Yaskawa INFORM job: R1_72,2(0,0)KM-OK.JBI

/JOB
//NAME R1_72,2(0,0)KM-OK
///FOLDERNAME KRIS-SCIANA
//POS
///NPOS 76,76,0,3,0,0
///TOOL 0
///POSTYPE PULSE
///PULSE
C00000=-88252,73272,-8021,3471,94135,-39741
C00001=-196921,-21278,-79002,-15523,92407,23647
C00002=-191529,-10180,-72050,-27767,99083,38733
C00003=-191529,-10180,-72050,-27767,99083,38733
C00004=-206105,-1744,-8023,-24853,79126,31669
C00005=-210790,-9435,-14216,-24034,77614,30226
C00006=-211112,-7151,-9678,-24113,76035,30431
C00007=-211112,-6884,-8412,-24172,75449,30554
C00008=-211112,-7143,-9634,-24115,76015,30436
C00009=-211447,-5344,-8192,-24050,75949,30323
C00010=-211112,-7143,-9634,-24115,76015,30436
C00011=-203899,-948,-19131,-24926,86387,30960
C00012=-203899,16721,-46212,-27001,109725,25798
C00013=-213997,-36135,-90156,-18508,92135,33607
C00014=-215703,-40125,-89891,-17749,89721,33477
C00015=-216394,-41642,-89732,-17450,88761,33414
C00016=-216190,-46458,-89537,-17546,86322,33825
C00017=-216581,-43974,-88082,-17376,86615,33666
C00018=-216757,-44589,-88447,-17302,86492,33627
C00019=-216394,-41642,-89732,-17450,88761,33414
C00020=-215410,-41044,-89232,-17867,88937,33676
C00021=-215562,-42319,-88713,-17803,87979,33772
C00022=-215410,-41044,-89232,-17867,88937,33676
C00023=-216394,-41642,-89732,-17450,88761,33414
C00024=-200348,-21688,-81312,-31633,113980,39480
C00025=-200646,-25016,-80489,-31008,111986,39985
C00026=-201612,-26033,-81353,-30788,111712,39736
C00027=-200646,-25016,-80489,-31008,111986,39985
C00028=-200348,-21688,-81312,-31633,113980,39480
C00029=-204378,-25649,-84759,-30672,112905,38454
C00030=-203466,-23371,-84449,-31149,114010,38425
C00031=-201237,-17494,-83481,-32404,116710,38313
C00032=-183775,-3850,-69382,-22164,99452,52082
C00033=-187139,105474,25900,5524,97478,-74523
C00034=-183987,78008,14988,-30780,97915,-53143
C00035=-185860,79679,21494,-38294,98804,-45722
C00036=-187540,86449,24962,5600,88344,-75041
C00037=-187072,89119,27221,5424,88298,-74904
C00038=-185446,79208,21072,-38405,98978,-45626
C00039=-185286,79610,21498,-38440,98994,-45572
C00040=-184095,83249,26388,-38603,98564,-44953
C00041=-184985,79410,21976,-38469,98802,-45386
C00042=-185085,78027,18507,-38623,99890,-45822
C00043=-184563,78672,15161,-39118,101977,-46400
C00044=-123480,133166,88670,-6552,116959,-64608
C00045=-123480,133166,88670,-6552,116959,-64608
C00046=-92269,117134,36709,3424,120351,-70294
C00047=-88374,116940,55217,-2527,120928,-72150
C00048=-88375,114548,55776,-2482,119356,-72114
C00049=-88651,123794,71043,-488,118252,-71721
C00050=-88408,114754,56297,-2480,119142,-72120
C00051=-88628,116331,59860,-2466,117754,-72169
C00052=-88954,122720,69576,-537,118600,-71834
C00053=-90233,119037,64628,-750,119747,-72317
C00054=-98563,95834,34419,17716,116287,-71642
C00055=-98641,94945,33315,17755,116515,-71636
C00056=-98178,89163,25359,18092,118260,-71172
C00057=-93588,99005,30718,8872,122903,-71358
C00058=-94574,131390,74567,2575,121590,-32143
C00059=-94435,131728,75046,2064,81257,-32153
C00060=-94150,154511,102675,2539,39785,-31487
C00061=-125444,148323,76798,-7366,54308,24231
C00062=-94150,154507,102675,2551,39784,-31488
C00063=-139725,-91160,-117526,-40600,105870,54843
C00064=-191529,-10180,-72050,-27767,99083,38733
C00065=-206105,-1744,-8023,-24853,79126,31669
C00066=-208371,-7084,-12355,-24468,78381,30975
C00067=-208875,-4028,-7246,-24508,76793,31119
C00068=-211010,-1092,-5442,-21718,78200,30111
C00069=-214621,-3970,-7511,-21112,77073,28985
C00070=-213962,-6039,-9919,-21200,77633,29128
C00071=-208371,-7084,-12355,-24468,78381,30975
C00072=-191529,-10180,-72050,-27767,99083,38733
C00073=-132846,-97761,-120048,-41164,107386,57132
C00074=-122033,25891,-66087,-31414,115477,22633
C00075=8893,25891,-66087,-31414,115477,22633
BC00000=280970,864873,1070899
BC00001=364125,1161342,1070909
BC00002=350007,1191142,1070910
BC00003=363568,1191142,637995
BC00004=363568,1191142,637995
BC00005=363568,1191142,637995
BC00006=363568,1191142,637995
BC00007=363568,1191142,637995
BC00008=363568,1191142,637995
BC00009=363568,1191142,637995
BC00010=363568,1191142,637995
BC00011=363568,1191142,637995
BC00012=363568,1191142,1070910
BC00013=350007,1191142,1070910
BC00014=344488,1191142,1070910
BC00015=342281,1191142,1070910
BC00016=339895,1191142,1070910
BC00017=339895,1191142,1070910
BC00018=342284,1191142,1070910
BC00019=342281,1191142,1070910
BC00020=336125,1191142,1070910
BC00021=336126,1191142,1070910
BC00022=336125,1191142,1070910
BC00023=342281,1191142,1070910
BC00024=300691,1191142,1070910
BC00025=300694,1191142,1070910
BC00026=300713,1191142,1070910
BC00027=300694,1191142,1070910
BC00028=300691,1191142,1070910
BC00029=314396,1191142,1070910
BC00030=315717,1191142,1070910
BC00031=319021,1191142,1070910
BC00032=331167,1109440,1070910
BC00033=374140,996980,1070910
BC00034=390851,1051981,1070910
BC00035=396168,1069059,1070910
BC00036=374323,999430,1070910
BC00037=374323,999430,1070910
BC00038=396168,1069059,1070910
BC00039=396168,1069059,1070910
BC00040=396168,1069059,1070910
BC00041=396168,1074643,1070910
BC00042=396168,1074757,1070910
BC00043=396168,1075043,1070910
BC00044=233365,1008921,1070910
BC00045=14833,1008921,1070910
BC00046=11006,981483,1070910
BC00047=11006,981483,1070910
BC00048=11729,977968,1070910
BC00049=12018,976562,1070910
BC00050=12018,976562,1070910
BC00051=12018,976562,1070910
BC00052=12018,976562,1070910
BC00053=12018,976562,1070910
BC00054=12018,976562,1070910
BC00055=12018,976562,1070910
BC00056=12018,976562,1070910
BC00057=12018,976562,1070910
BC00058=8338,956870,1070910
BC00059=8338,956870,1070910
BC00060=8339,956871,1070908
BC00061=260149,1038260,1070909
BC00062=325780,956871,1070907
BC00063=350007,1079161,1070910
BC00064=350007,1191142,1070910
BC00065=363568,1191142,637995
BC00066=363568,1191142,637995
BC00067=363568,1191142,637995
BC00068=363568,1191142,637995
BC00069=363568,1191142,637995
BC00070=363568,1191142,637995
BC00071=363568,1191142,637995
BC00072=350007,1191142,1070910
BC00073=350007,793911,1070910
BC00074=247929,729127,1070909
BC00075=145595,729127,1070909
///POSTYPE BASE
///RECTAN
///RCONF 0,0,0,0,0,0,0,0,0,0,0,0,0,0,0,0,0,0,0,0,0,0,0,0
P00006=0.222,-3.123,-1.508,0.0000,0.0000,0.0000
P00021=-0.225,-6.128,-0.405,0.0000,0.0000,0.0000
P00030=5.926,-4.294,-1.390,0.0000,0.0000,0.0000
//INST
///DATE 2024/07/30 11:04
///ATTR SC,RW
///GROUP1 RB1,BS1
NOP
'R1_72.2(0,0)
'Path S1563
SFTOF
MOVJ C00000 BC00000 VJ=100.00
MOVJ C00001 BC00001 VJ=100.00
MOVJ C00002 BC00002 VJ=70.00
MOVJ C00003 BC00003 VJ=70.00
MOVJ C00004 BC00004 VJ=70.00
MOVL C00005 BC00005 V=333.3
MOVL C00006 BC00006 V=166.7
REFP 3 C00007 BC00007
CALL JOB:SEARCH-R1
SET P030 P006
SFTON P030
MOVL C00008 BC00008 V=100.0
REFP 3 C00009 BC00009
CALL JOB:SEARCH-R1
SET P030 P006
SFTON P030
MOVL C00010 BC00010 V=100.0
SFTOF
MOVL C00011 BC00011 V=400.0
MOVL C00012 BC00012 V=1000.0
MOVJ C00013 BC00013 VJ=70.00
MOVJ C00014 BC00014 VJ=50.00
MOVL C00015 BC00015 V=100.0
MOVL C00016 BC00016 V=60.0
REFP 3 C00017 BC00017
CALL JOB:SEARCH-R1
SET P021 P006
SFTON P021
MOVL C00018 BC00018 V=60.0
MOVL C00019 BC00019 V=100.0
MOVL C00020 BC00020 V=60.0
REFP 3 C00021 BC00021
CALL JOB:SEARCH-R1
SET P021 P006
SFTON P021
MOVL C00022 BC00022 V=60.0
MOVL C00023 BC00023 V=100.0
MOVL C00024 BC00024 V=100.0
MOVL C00025 BC00025 V=60.0
REFP 3 C00026 BC00026
CALL JOB:SEARCH-R1
SET P021 P006
SFTON P021
MOVL C00027 BC00027 V=60.0
MOVL C00028 BC00028 V=100.0
MOVL C00029 BC00029 V=100.0
MOVL C00030 BC00030 V=166.7
MOVL C00031 BC00031 V=166.7
'Path VIA1564
SFTOF
MOVJ C00032 BC00032 VJ=50.00
'Path W1561
SFTOF
SFTON P021
MOVJ C00033 BC00033 VJ=50.00
MOVJ C00034 BC00034 VJ=100.00
SFTON P021
MOVL C00035 BC00035 V=166.7 PL=0
REFP 1 C00036 BC00036
REFP 2 C00037 BC00037
MACRO1 MJ#(0) ARGF6
ARCON
MOVL C00038 BC00038 V=10.8
MOVL C00039 BC00039 V=10.8
MOVL C00040 BC00040 V=10.8
MOVL C00041 BC00041 V=10.8
ARCOF
MOVL C00042 BC00042 V=100.0
MOVL C00043 BC00043 V=166.7
SFTOF
'Path VIA1565
SFTOF
MOVJ C00044 BC00044 VJ=50.00
MOVJ C00045 BC00045 VJ=50.00
'Path W1566
SFTOF
SFTON P021
MOVJ C00046 BC00046 VJ=100.00
MOVJ C00047 BC00047 VJ=100.00
MOVJ C00048 BC00048 VJ=50.00
MOVL C00049 BC00049 V=100.0 PL=0
REFP 1 C00050 BC00050
REFP 2 C00051 BC00051
MACRO1 MJ#(0) ARGF5
ARCON
MOVL C00052 BC00052 V=8.3
MOVL C00053 BC00053 V=8.3
ARCOF
MOVL C00054 BC00054 V=10.0
ARCON
MOVL C00055 BC00055 V=8.3
MOVL C00056 BC00056 V=8.3
ARCOF
MOVL C00057 BC00057 V=166.7
MOVL C00058 BC00058 V=333.3
SFTOF
MOVJ C00059 BC00059 VJ=50.00
MOVJ C00060 BC00060 VJ=100.00
MOVJ C00061 BC00061 VJ=70.00
MOVL C00062 BC00062 V=1000.0
MOVJ C00063 BC00063 VJ=70.00
MOVJ C00064 BC00064 VJ=70.00
MOVJ C00065 BC00065 VJ=70.00
MOVL C00066 BC00066 V=333.3
SFTON P030
MOVL C00067 BC00067 V=166.7
MOVL C00068 BC00068 V=100.0 PL=0
MACRO1 MJ#(0) ARGF7
ARCON
MOVL C00069 BC00069 V=9.2
ARCOF
MOVL C00070 BC00070 V=233.3
SFTOF
MOVL C00071 BC00071 V=333.3
MOVL C00072 BC00072 V=666.7
MOVJ C00073 BC00073 VJ=70.00
MOVJ C00074 BC00074 VJ=70.00
MOVJ C00075 BC00075 VJ=100.00
END
